% RSLogix 500 project PROC1_PID_CONTROL.RSS, saved by version 8.30.00.16 %
PROJECT "PROC1"    % processor: Bul.1763 MicroLogix 1100 Series B %

PROGRAM FILES
  LAD 2   5 rungs

DATA FILES
  O0 OUTPUT  4 elements
  I1 INPUT  6 elements
  S2 STATUS  66 elements
  B3 BINARY  1 elements
  T4 TIMER  1 elements
  C5 COUNTER  1 elements
  R6 CONTROL  1 elements
  N7 INTEGER  21 elements
  F8 FLOAT  1 elements
  PD22   1 elements

LADDER 2
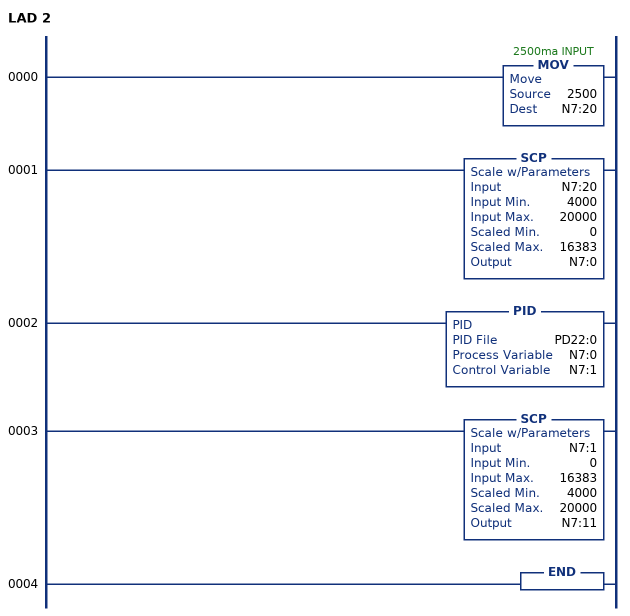
% Rung: 0 %
SOR MOV 2500 N7:20 EOR
%   N7:20  "2500ma INPUT" %
% Rung: 1 %
SOR SCP N7:20 4000 20000 0 16383 N7:0 EOR
%   N7:20  "2500ma INPUT" %
% Rung: 2 %
SOR PID PD22:0 N7:0 N7:1 EOR
% Rung: 3 %
SOR SCP N7:1 0 16383 4000 20000 N7:11 EOR
% Rung: 4 %
SOR END EOR
